// LS Electric XG5000 project: 16-38-1
// PLC NewPLC
// module base 0 slot 0: 입출력 모듈:XBC-DR14E (DC 24V 입력 8점, 릴레이 출력 6점)

PROGRAM NewProgram (task: 스캔 프로그램)

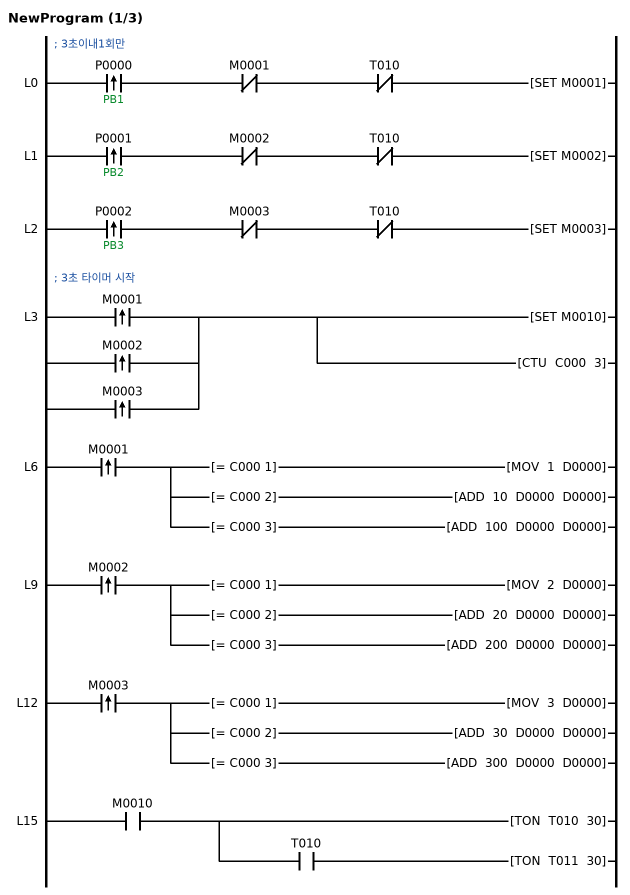
; L0
LOADP     P0000	// PB1
AND NOT   M0001
AND NOT   T010
SET       M0001
// output comment: 3초이내1회만
; L1
LOADP     P0001	// PB2
AND NOT   M0002
AND NOT   T010
SET       M0002
; L2
LOADP     P0002	// PB3
AND NOT   M0003
AND NOT   T010
SET       M0003
; L3
LOADP     M0001
ORP       M0002
ORP       M0003
SET       M0010
CTU       C000 3
// output comment: 3초 타이머 시작
; L6
LOADP     M0001
MPUSH
AND=      C000 1
MOV       1 D0000
MLOAD
AND=      C000 2
ADD       10 D0000 D0000
MPOP
AND=      C000 3
ADD       100 D0000 D0000
; L9
LOADP     M0002
MPUSH
AND=      C000 1
MOV       2 D0000
MLOAD
AND=      C000 2
ADD       20 D0000 D0000
MPOP
AND=      C000 3
ADD       200 D0000 D0000
; L12
LOADP     M0003
MPUSH
AND=      C000 1
MOV       3 D0000
MLOAD
AND=      C000 2
ADD       30 D0000 D0000
MPOP
AND=      C000 3
ADD       300 D0000 D0000
; L15
LOAD      M0010
TON       T010 30
AND       T010
TON       T011 30

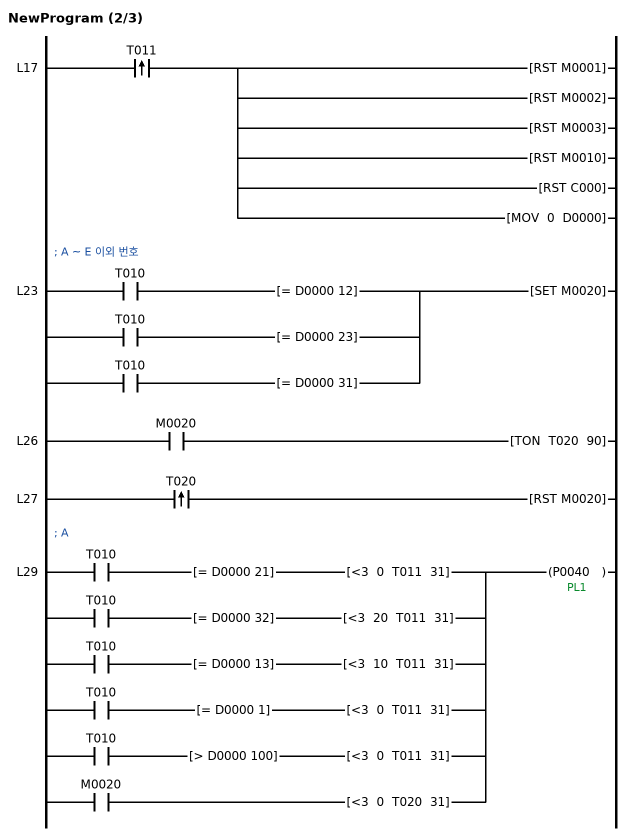
; L17
LOADP     T011
RST       M0001
RST       M0002
RST       M0003
RST       M0010
RST       C000
MOV       0 D0000
; L23
LOAD      T010
AND=      D0000 12
LOAD      T010
AND=      D0000 23
OR LOAD
LOAD      T010
AND=      D0000 31
OR LOAD
SET       M0020
// output comment: A ~ E 이외 번호
; L26
LOAD      M0020
TON       T020 90
; L27
LOADP     T020
RST       M0020
; L29
LOAD      T010
AND=      D0000 21
AND<3     0 T011 31
LOAD      T010
AND=      D0000 32
AND<3     20 T011 31
OR LOAD
LOAD      T010
AND=      D0000 13
AND<3     10 T011 31
OR LOAD
LOAD      T010
AND=      D0000 1
AND<3     0 T011 31
OR LOAD
LOAD      T010
AND>      D0000 100
AND<3     0 T011 31
OR LOAD
LOAD      M0020
AND<3     0 T020 31
OR LOAD
OUT       P0040	// PL1
// output comment: A

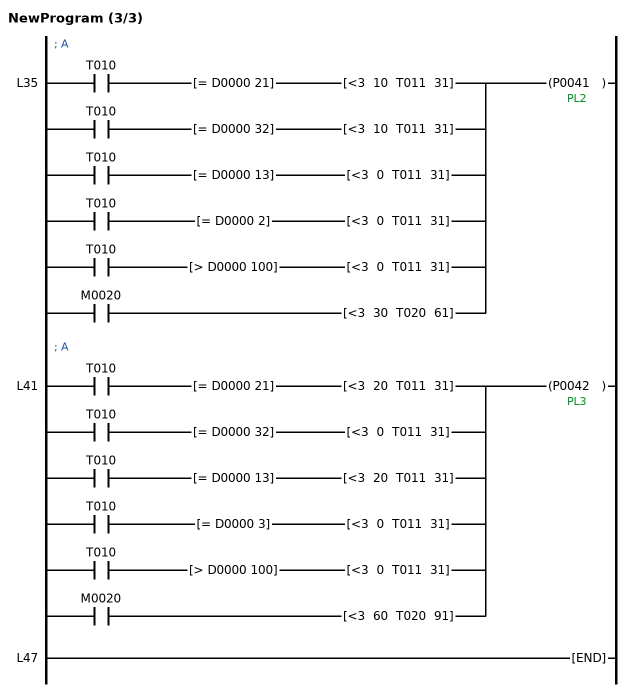
; L35
LOAD      T010
AND=      D0000 21
AND<3     10 T011 31
LOAD      T010
AND=      D0000 32
AND<3     10 T011 31
OR LOAD
LOAD      T010
AND=      D0000 13
AND<3     0 T011 31
OR LOAD
LOAD      T010
AND=      D0000 2
AND<3     0 T011 31
OR LOAD
LOAD      T010
AND>      D0000 100
AND<3     0 T011 31
OR LOAD
LOAD      M0020
AND<3     30 T020 61
OR LOAD
OUT       P0041	// PL2
// output comment: A
; L41
LOAD      T010
AND=      D0000 21
AND<3     20 T011 31
LOAD      T010
AND=      D0000 32
AND<3     0 T011 31
OR LOAD
LOAD      T010
AND=      D0000 13
AND<3     20 T011 31
OR LOAD
LOAD      T010
AND=      D0000 3
AND<3     0 T011 31
OR LOAD
LOAD      T010
AND>      D0000 100
AND<3     0 T011 31
OR LOAD
LOAD      M0020
AND<3     60 T020 91
OR LOAD
OUT       P0042	// PL3
// output comment: A
; L47
END